//==================================================================================================
//							Beckhoff Automation Poland
//									23.05.2017
//	Struktura zawierajaca definicje zdarzenia
// 	v1.0	|| TC v 3.1.4020.32		|| - pierwsza wersja
//==================================================================================================
TYPE ST_EventDefinition :
STRUCT
	dwClass									: DWORD;
	dwParam									: DWORD;
	wsMessage								: WSTRING(80);
	bActive									: BOOL;
END_STRUCT
END_TYPE

(* stored: Version 1.1.0.1, ProductVersion 3.1.4020.12
   DUT ST_EventDefinition: Id {abb9c617-5f0d-430b-8f5a-2b7f281d0205} *)
